Yaskawa INFORM job: R1_W27-A2(90,-90)POPR-KM-OK.JBI

/JOB
//NAME R1_W27-A2(90,-90)POPR-KM-OK
///FOLDERNAME KRIS-SCIANA
//POS
///NPOS 176,176,0,6,0,0
///TOOL 0
///POSTYPE PULSE
///PULSE
C00000=-47255,94033,21850,39667,98426,-85112
C00001=-10855,-90146,-90520,33531,76579,-85488
C00002=111602,-139984,-127808,5509,79015,30630
C00003=111602,-139984,-127808,5509,79015,30630
C00004=63451,-100439,-89596,34729,108559,18896
C00005=79235,-88636,-73634,36549,98880,22423
C00006=81155,-89027,-70716,36576,96440,22410
C00007=83679,-91038,-71523,36826,94925,22960
C00008=83320,-90762,-71414,36792,95139,22882
C00009=83320,-91266,-72707,36833,95574,23028
C00010=84421,-92107,-73039,36936,94918,23269
C00011=84421,-91766,-72172,36910,94628,23171
C00012=81728,-90820,-74480,36776,97327,22951
C00013=111602,-139984,-127808,5509,79015,30630
C00014=111602,-139984,-127808,5509,79015,30630
C00015=131748,-141997,-126846,-10495,77447,36936
C00016=120565,-130076,-92733,-8792,61450,34172
C00017=114295,-129242,-91918,-7183,60764,31836
C00018=112834,-127676,-89826,-6827,60159,31317
C00019=109595,-127191,-89697,-5944,60074,30085
C00020=111525,-128681,-91514,-6443,60572,30793
C00021=111525,-130307,-93896,-6407,61199,30757
C00022=120936,-129452,-91830,-16171,61520,34917
C00023=118478,-129412,-91819,-15577,61061,34026
C00024=114109,-131661,-95461,-7074,61680,31708
C00025=125724,-139860,-107023,-9755,65762,35760
C00026=168598,-161440,-97829,-65849,65951,-5239
C00027=139953,-89870,-86584,-36793,78283,-52428
C00028=129963,-49074,-62936,-33723,79499,-56916
C00029=128367,-48213,-57426,-33587,76404,-56612
C00030=128171,-46376,-53454,-33725,75068,-56281
C00031=127551,-46486,-53520,-33557,74812,-56456
C00032=127838,-49102,-55957,-33615,75055,-56414
C00033=127838,-49096,-59569,-33337,76927,-56985
C00034=130300,-24150,-34218,-41893,86298,-55823
C00035=130416,-25931,-34035,-41938,85581,-55484
C00036=130524,-27637,-35221,-41959,85519,-55412
C00037=130416,-25931,-34035,-41938,85581,-55484
C00038=129161,-28892,-39611,-41713,86429,-56383
C00039=125861,-39018,-45021,-41293,83456,-56659
C00040=125861,-38957,-44315,-41317,83150,-56538
C00041=125861,-39018,-45021,-41293,83456,-56659
C00042=132006,-10593,-25804,-42105,88453,-55942
C00043=125383,-9861,-27484,-30967,87136,-57090
C00044=124817,-9932,-27539,-30868,86930,-57252
C00045=125341,-12485,-30902,-30958,87772,-57281
C00046=124961,-12409,-32279,-30889,88403,-57596
C00047=121984,-15512,-34257,-30384,87021,-58359
C00048=122055,-13679,-30637,-30418,85927,-58040
C00049=122041,-11816,-29206,-30415,85989,-58061
C00050=122055,-13679,-30637,-30418,85927,-58040
C00051=122071,-15599,-34612,-30398,87201,-58373
C00052=118054,-13550,-32366,-29609,85516,-59451
C00053=118054,-13583,-31956,-29617,85281,-59389
C00054=118054,-13550,-32366,-29609,85516,-59451
C00055=125534,-18569,-39431,-41052,88700,-58862
C00056=123834,-57988,-65399,-23223,94284,39293
C00057=119710,-36131,-50756,-23492,104469,35737
C00058=119541,-35148,-48081,-23365,103369,35899
C00059=120820,-55138,-59718,-22945,91575,38721
C00060=119503,-55193,-60983,-22866,91905,38180
C00061=118759,-58952,-61759,-21710,87152,34499
C00062=120697,-55018,-60828,-22957,92227,38551
C00063=123778,-56814,-67966,-23331,96280,38880
C00064=80812,-71471,-83715,15937,85664,-13866
C00065=80812,-71834,-71790,16172,78419,-14815
C00066=107747,-97676,-64864,-15422,34839,20449
C00067=107974,-98087,-64546,-15779,34491,20660
C00068=108174,-97847,-63422,-16183,33983,20896
C00069=108174,-97847,-63422,-16183,33983,20896
C00070=109575,-108888,-72439,-17471,34149,21710
C00071=102046,-72347,-67920,-1263,67597,24279
C00072=76953,-69983,-67153,17125,77381,-16337
C00073=77709,-68021,-67434,16896,78355,-15929
C00074=96304,-74836,-69045,2706,67540,13944
C00075=85382,-70192,-66839,14096,72335,1446
C00076=83671,-68641,-66151,14549,72999,911
C00077=82927,-72320,-69596,14740,73354,686
C00078=82383,-44408,-60013,10514,90636,-51553
C00079=83267,-39109,-54206,10352,89686,-51335
C00080=93739,1438,-24878,6422,91479,-57500
C00081=93739,1438,-24878,6422,91479,-57500
C00082=93483,1925,-29171,6495,94374,-57435
C00083=103631,8716,-24589,-7355,104161,-72543
C00084=103148,15486,-14064,-7496,103326,-72736
C00085=105595,14163,-15273,-7551,103608,-71922
C00086=104864,13485,-18488,-6736,105180,-72257
C00087=101225,7871,-25887,-447,100429,-73560
C00088=94829,-40669,-100015,6490,88409,-74102
C00089=128133,-139556,-106944,-10306,66166,36618
C00090=113623,-140124,-95696,-7245,57468,31798
C00091=111191,-133211,-91671,-6501,58335,30798
C00092=112396,-117188,-87436,-6483,64023,30924
C00093=117788,-123916,-92276,-7889,64025,32937
C00094=117788,-143811,-128922,-7332,76251,32157
C00095=117788,-143811,-128922,-7332,76251,32157
C00096=-27890,68892,-2811,-32304,95656,-64919
C00097=-1389,132560,29341,8972,98096,-84314
C00098=-17183,121165,41486,39124,87360,-83411
C00099=45609,12223,-14680,25874,102540,-44378
C00100=55301,17182,-10314,25374,99523,-41463
C00101=55301,16672,-6013,25146,96878,-42036
C00102=55301,16639,-5464,25122,96557,-42106
C00103=55301,16672,-6013,25146,96878,-42036
C00104=52027,31709,8447,25239,96790,-43264
C00105=65662,27936,-1686,1783,97311,-42028
C00106=65925,27175,-1528,1759,96817,-41946
C00107=66144,26660,-2030,1742,96856,-41873
C00108=65925,27175,-1528,1759,96817,-41946
C00109=65925,27520,-3302,1766,98087,-41928
C00110=67752,27932,-3186,1610,98190,-41320
C00111=69686,29368,267,1433,96766,-40698
C00112=69239,27811,-1265,1472,96915,-40843
C00113=69714,29591,-377,1432,97275,-40681
C00114=70571,32771,2169,1358,97331,-40400
C00115=72811,38961,10399,1155,95415,-39677
C00116=73243,40763,12275,1116,95181,-39535
C00117=72717,38685,9237,1163,95989,-39704
C00118=70300,45171,15024,1377,95797,-40506
C00119=71840,46165,18079,1239,94403,-40008
C00120=72279,45156,17000,1201,94542,-39861
C00121=71840,46165,18079,1239,94403,-40008
C00122=71100,43306,13055,1308,96038,-40237
C00123=74981,35157,4595,968,97003,-38944
C00124=68153,50345,23565,13015,101581,-39746
C00125=68153,50336,23863,13003,101398,-39766
C00126=68153,50345,23565,13015,101581,-39746
C00127=74981,36365,46,979,100422,-38916
C00128=68608,6976,-17792,23795,112053,-53591
C00129=69057,8041,-13956,23524,110262,-53802
C00130=77166,501,-24156,13228,105180,-53608
C00131=69228,8608,-13543,23550,110248,-53738
C00132=68547,9857,-11185,23337,109691,-54121
C00133=80532,13332,-12849,13354,104269,-52437
C00134=69002,6644,-20376,25626,106012,-45957
C00135=36743,66838,47163,37250,103366,-40352
C00136=37959,59579,46469,37755,95211,-37788
C00137=37837,59881,47347,37721,94956,-37928
C00138=37624,60339,48596,37673,94623,-38135
C00139=36831,72187,58039,36474,100818,-41891
C00140=49145,73657,39688,12770,111067,-36167
C00141=47533,6238,-21702,16193,87850,-22319
C00142=48706,7477,-14718,15969,84101,-22409
C00143=50440,12407,-9463,15589,83099,-21944
C00144=49368,8705,-13714,15818,83988,-22197
C00145=48664,7312,-13691,15994,83418,-22513
C00146=49682,14586,-7490,15763,83149,-22198
C00147=45719,31490,8640,21979,89950,-33295
C00148=45824,34631,11803,21965,89613,-33319
C00149=48704,7662,-16449,15949,85218,-22264
C00150=47002,4841,-19925,16324,86209,-22716
C00151=51620,13344,-12650,-10356,82695,15963
C00152=52172,14147,-8973,-10543,80943,16297
C00153=53042,17284,-5127,-10797,80314,16646
C00154=52937,12849,-8980,-10764,80389,16602
C00155=52386,14618,-8611,-10600,80988,16365
C00156=54599,19555,-5413,-11177,81839,17037
C00157=52866,15720,-8829,-10712,81740,16462
C00158=52320,14787,-11359,-10544,82730,16194
C00159=103684,1413,-30862,2741,121345,77818
C00160=103850,2833,-28631,2757,120697,77864
C00161=102574,7420,-23963,2468,120223,77363
C00162=103907,3755,-28694,2786,121208,77898
C00163=104106,5504,-25931,2802,120401,77953
C00164=105308,5972,-25223,3052,120166,78404
C00165=104815,6248,-27488,2999,121717,78261
C00166=103683,1405,-30869,2741,121346,77818
C00167=103614,2055,-30742,3606,100061,77951
C00168=110138,-139455,-127658,5821,79297,30141
C00169=62576,-99046,-89073,34649,109242,18742
C00170=76661,-93546,-74524,35984,98364,21158
C00171=71402,-81532,-60843,44640,104085,20726
C00172=76616,-70399,-55778,46201,103281,22914
C00173=72927,-70202,-57613,45814,106055,22410
C00174=72965,-71329,-91142,53207,119453,30086
C00175=-4535,-93265,-111062,3717,101159,77715
BC00000=172948,1022366,1065683
BC00001=284631,1066333,1053590
BC00002=197512,1190309,1009585
BC00003=397680,1190309,1009585
BC00004=397680,1190309,1009585
BC00005=397680,1190309,1009585
BC00006=397680,1190309,1009585
BC00007=397680,1190309,1009585
BC00008=397680,1190309,1009585
BC00009=397680,1190309,1009585
BC00010=397680,1190309,1009585
BC00011=397680,1190309,1009585
BC00012=397680,1190309,1009585
BC00013=397680,1190309,1009585
BC00014=197512,1190309,1009585
BC00015=15680,1190309,1003705
BC00016=15680,1190309,1003705
BC00017=15680,1190309,1003705
BC00018=15680,1190309,1003705
BC00019=15680,1190309,1003705
BC00020=15680,1190309,1003705
BC00021=15680,1190309,1003705
BC00022=15680,1190309,1003705
BC00023=15680,1190309,1003705
BC00024=15680,1190309,1003705
BC00025=15680,1190309,1003705
BC00026=2250,1188982,1018188
BC00027=2245,1185181,1042831
BC00028=2245,1185181,1042831
BC00029=2245,1185181,1042831
BC00030=2245,1185181,1042831
BC00031=2245,1185181,1042831
BC00032=2245,1185181,1042831
BC00033=2245,1185181,1042831
BC00034=1991,1180873,1070755
BC00035=1991,1180873,1070755
BC00036=1991,1180873,1070755
BC00037=1991,1180873,1070755
BC00038=1991,1180873,1070755
BC00039=1991,1180873,1070755
BC00040=1991,1180873,1070755
BC00041=1991,1180873,1070755
BC00042=1991,1180873,1070755
BC00043=1991,1180873,1070755
BC00044=1991,1180873,1070755
BC00045=1991,1180873,1070755
BC00046=1991,1180873,1070755
BC00047=1991,1180873,1070755
BC00048=1991,1180873,1070755
BC00049=1991,1180873,1070755
BC00050=1991,1180873,1070755
BC00051=1991,1180873,1070755
BC00052=1991,1180873,1070755
BC00053=1991,1180873,1070755
BC00054=1991,1180873,1070755
BC00055=1991,1180873,1070755
BC00056=1991,1143594,1070910
BC00057=1991,1145344,1070910
BC00058=1991,1145344,1070910
BC00059=1991,1145344,1070910
BC00060=1991,1145344,1070910
BC00061=1991,1130616,1070910
BC00062=1991,1130116,1070910
BC00063=1991,1128866,1070910
BC00064=1991,1180480,1070910
BC00065=1991,1180480,1070910
BC00066=1992,1180480,1070906
BC00067=1992,1180480,1070906
BC00068=1992,1180480,1070906
BC00069=1992,1180480,1070906
BC00070=1992,1180480,1070906
BC00071=1992,1180480,1070906
BC00072=1991,1175938,1070910
BC00073=1991,1175938,1070910
BC00074=1992,1180480,1070906
BC00075=1992,1180480,1070906
BC00076=1992,1180480,1070906
BC00077=1992,1180480,1070906
BC00078=1992,1180480,1070906
BC00079=1993,1180480,1070905
BC00080=1992,1180480,1070906
BC00081=1992,1180480,1070906
BC00082=1992,1180480,1070906
BC00083=1993,1170260,1070904
BC00084=1993,1170260,1070902
BC00085=1993,1170260,1070902
BC00086=1993,1170260,1070904
BC00087=1992,1180480,1070906
BC00088=1992,1180480,1070906
BC00089=18069,1190309,1003705
BC00090=18069,1190309,1003705
BC00091=18069,1190309,1003705
BC00092=18069,1190309,1003705
BC00093=18069,1190309,1003705
BC00094=18069,1190309,1003705
BC00095=94851,1192591,1003705
BC00096=27006,1176774,1055878
BC00097=57075,1322294,1070892
BC00098=45628,1277740,1070896
BC00099=248889,1187650,1070910
BC00100=248889,1187650,1070910
BC00101=248889,1187650,1070910
BC00102=248889,1187650,1070910
BC00103=248889,1187650,1070910
BC00104=248889,1187650,1070910
BC00105=248889,1187650,1070910
BC00106=248889,1187650,1070910
BC00107=248889,1187650,1070910
BC00108=248889,1187650,1070910
BC00109=248889,1187650,1070910
BC00110=248889,1187650,1070910
BC00111=248889,1187650,1070910
BC00112=248889,1187650,1070910
BC00113=248889,1187650,1070910
BC00114=248889,1187650,1070910
BC00115=248889,1187650,1070910
BC00116=248889,1187650,1070910
BC00117=248889,1187650,1070910
BC00118=248889,1187650,1070910
BC00119=248889,1187650,1070910
BC00120=248889,1187650,1070910
BC00121=248889,1187650,1070910
BC00122=248889,1187650,1070910
BC00123=248889,1187650,1070910
BC00124=248889,1187650,1070910
BC00125=248889,1187650,1070910
BC00126=248889,1187650,1070910
BC00127=248889,1187650,1070910
BC00128=312191,1167362,1070910
BC00129=306535,1168545,1070910
BC00130=306538,1168544,1070910
BC00131=304272,1169019,1070910
BC00132=304272,1169019,1070910
BC00133=306538,1168544,1070910
BC00134=306535,1168545,1070910
BC00135=199299,1192678,1070910
BC00136=199299,1192678,1070910
BC00137=199299,1192678,1070910
BC00138=199299,1192678,1070910
BC00139=199299,1192678,1070910
BC00140=199299,1192678,1070910
BC00141=199962,1192678,1070910
BC00142=199962,1192678,1070910
BC00143=199962,1192678,1070910
BC00144=200228,1192678,1070910
BC00145=200228,1192678,1070910
BC00146=199962,1192678,1070910
BC00147=199962,1192678,1070910
BC00148=199962,1192678,1070910
BC00149=202074,1192678,1070910
BC00150=201410,1192678,1070910
BC00151=150763,1159292,1070910
BC00152=156327,1160542,1070910
BC00153=158126,1160946,1070907
BC00154=158552,1161042,1070910
BC00155=158552,1161042,1070910
BC00156=158692,1122943,1055155
BC00157=156466,1122443,1062648
BC00158=150903,1121193,1070910
BC00159=346682,1128113,1048282
BC00160=345916,1134373,1032919
BC00161=345708,1136079,1028733
BC00162=345610,1136877,1026774
BC00163=345610,1136877,1026774
BC00164=345708,1136079,1028733
BC00165=345610,1136877,1026774
BC00166=343614,1128095,1048354
BC00167=343613,1128096,1048352
BC00168=396087,1032525,1009585
BC00169=396087,1190309,1009585
BC00170=396087,1190309,1009585
BC00171=396087,1190309,1009585
BC00172=396087,1190309,1009585
BC00173=396087,1190309,1009585
BC00174=396087,1190309,1009585
BC00175=174979,687379,1048352
///POSTYPE BASE
///RECTAN
///RCONF 0,0,0,0,0,0,0,0,0,0,0,0,0,0,0,0,0,0,0,0,0,0,0,0
P00006=0.222,-3.123,-1.508,0.0000,0.0000,0.0000
P00023=0.143,-0.036,0.682,0.0000,0.0000,0.0000
P00024=0.145,-0.552,1.326,0.0000,0.0000,0.0000
P00025=-2.003,0.006,0.728,0.0000,0.0000,0.0000
P00040=-0.030,9.648,2.467,0.0000,0.0000,0.0000
P00041=0.192,3.924,0.305,0.0000,0.0000,0.0000
//INST
///DATE 2024/07/23 11:10
///ATTR SC,RW
///GROUP1 RB1,BS1
NOP
SFTOF
MOVJ C00000 BC00000 VJ=100.00
MOVJ C00001 BC00001 VJ=100.00
MOVJ C00002 BC00002 VJ=100.00
'DODANO BP 060624
MOVJ C00003 BC00003 VJ=100.00
MOVJ C00004 BC00004 VJ=100.00
MOVL C00005 BC00005 V=233.3
MOVL C00006 BC00006 V=60.0
REFP 3 C00007 BC00007
CALL JOB:SEARCH-R1
SET P040 P006
SFTON P040
MOVL C00008 BC00008 V=100.0
MOVL C00009 BC00009 V=100.0
MOVL C00010 BC00010 V=60.0
REFP 3 C00011 BC00011
CALL JOB:SEARCH-R1
SET P040 P006
SFTON P040
MOVL C00012 BC00012 V=100.0
SFTOF
MOVJ C00013 BC00013 VJ=100.00
MOVJ C00014 BC00014 VJ=100.00
MOVL C00015 BC00015 V=666.7
MOVL C00016 BC00016 V=666.7
MOVL C00017 BC00017 V=233.3
MOVL C00018 BC00018 V=60.0
REFP 3 C00019 BC00019
CALL JOB:SEARCH-R1
SET P041 P006
SFTON P041
MOVL C00020 BC00020 V=100.0
MOVL C00021 BC00021 V=100.0
MOVL C00022 BC00022 V=60.0
REFP 3 C00023 BC00023
CALL JOB:SEARCH-R1
SET P041 P006
SFTON P041
MOVL C00024 BC00024 V=100.0
MOVL C00025 BC00025 V=666.7
'KONIEC BP 060624
MOVJ C00026 BC00026 VJ=100.00
MOVJ C00027 BC00027 VJ=100.00
MOVJ C00028 BC00028 VJ=100.00
MOVJ C00029 BC00029 VJ=100.00
MOVL C00030 BC00030 V=60.0
REFP 3 C00031 BC00031
CALL JOB:SEARCH-R1
SET P023 P006
SFTON P023
MOVL C00032 BC00032 V=60.0
MOVL C00033 BC00033 V=100.0
MOVL C00034 BC00034 V=100.0
MOVL C00035 BC00035 V=100.0
REFP 3 C00036 BC00036
CALL JOB:SEARCH-R1
SET P023 P006
SFTON P023
MOVL C00037 BC00037 V=60.0
MOVL C00038 BC00038 V=100.0
MOVL C00039 BC00039 V=100.0
REFP 3 C00040 BC00040
CALL JOB:SEARCH-R1
SET P023 P006
SFTON P023
MOVL C00041 BC00041 V=60.0
'DRUGI NOWY POMIAR
SFTOF
MOVL C00042 BC00042 V=100.0
MOVL C00043 BC00043 V=100.0
REFP 3 C00044 BC00044
CALL JOB:SEARCH-R1
SET P024 P006
SFTON P024
MOVL C00045 BC00045 V=60.0
MOVL C00046 BC00046 V=100.0
MOVL C00047 BC00047 V=100.0
MOVL C00048 BC00048 V=60.0
REFP 3 C00049 BC00049
CALL JOB:SEARCH-R1
SET P024 P006
SFTON P024
MOVL C00050 BC00050 V=60.0
MOVL C00051 BC00051 V=100.0
MOVL C00052 BC00052 V=60.0
REFP 3 C00053 BC00053
CALL JOB:SEARCH-R1
SET P024 P006
SFTON P024
MOVL C00054 BC00054 V=60.0
MOVJ C00055 BC00055 VJ=30.00
SFTOF
'Path W988
SFTOF
SFTON P023
MOVJ C00056 BC00056 VJ=50.00
MOVJ C00057 BC00057 VJ=100.00
MOVL C00058 BC00058 V=100.0 PL=0
REFP 1 C00059 BC00059
REFP 2 C00060 BC00060
MACRO1 MJ#(0) ARGF7
ARCON
SFTON P024
MOVL C00061 BC00061 V=10.8
ARCOF
MOVL C00062 BC00062 V=100.0
MOVJ C00063 BC00063 VJ=50.00
SFTOF
'Path W989
SFTOF
SFTON P023
MOVJ C00064 BC00064 VJ=100.00
MOVJ C00065 BC00065 VJ=50.00
MOVL C00066 BC00066 V=100.0
ARCON
MOVL C00067 BC00067 V=8.3
MOVL C00068 BC00068 V=8.3
MOVL C00069 BC00069 V=8.3
ARCOF
SFTOF
MOVL C00070 BC00070 V=83.3
SFTON P023
MOVL C00071 BC00071 V=100.0 PL=0
REFP 1 C00072 BC00072
REFP 2 C00073 BC00073
MACRO1 MJ#(0) ARGF7
ARCON
TIMER T=0.50
MOVL C00074 BC00074 V=10.0
MOVL C00075 BC00075 V=10.0
MOVL C00076 BC00076 V=10.0
ARCOF
MOVJ C00077 BC00077 VJ=15.00
MOVJ C00078 BC00078 VJ=100.00
SFTON P023
MOVJ C00079 BC00079 VJ=100.00
ARCON
SFTON P024
MOVL C00080 BC00080 V=10.0
MOVL C00081 BC00081 V=10.0
ARCOF
MOVJ C00082 BC00082 VJ=15.00
MOVJ C00083 BC00083 VJ=100.00
MOVJ C00084 BC00084 VJ=20.00
ARCON
MOVL C00085 BC00085 V=10.0
ARCOF
MOVL C00086 BC00086 V=100.0
MOVL C00087 BC00087 V=166.7
MOVJ C00088 BC00088 VJ=100.00
SFTOF
'BP 060624
MOVJ C00089 BC00089 VJ=100.00
MOVJ C00090 BC00090 VJ=100.00
SFTON P041
MOVL C00091 BC00091 V=100.0 PL=0
MACRO1 MJ#(0) ARGF6
ARCON
MOVL C00092 BC00092 V=12.5
ARCOF
MOVL C00093 BC00093 V=11.7
SFTOF
MOVL C00094 BC00094 V=666.7
MOVL C00095 BC00095 V=666.7
'KONIEC BP 060624
'2 STRONA
MOVJ C00096 BC00096 VJ=100.00
'Path VIA1124
SFTOF
MOVJ C00097 BC00097 VJ=100.00
CALL JOB:ONLY_CUT_KM_NEW_SCIANA
'Path S992
SFTOF
MOVJ C00098 BC00098 VJ=100.00
SFTOF
MOVJ C00099 BC00099 VJ=100.00
MOVJ C00100 BC00100 VJ=100.00
MOVL C00101 BC00101 V=133.3
REFP 3 C00102 BC00102
CALL JOB:SEARCH-R1
SET P024 P006
SFTON P024
MOVL C00103 BC00103 V=60.0
MOVL C00104 BC00104 V=100.0
MOVL C00105 BC00105 V=100.0
MOVL C00106 BC00106 V=100.0
REFP 3 C00107 BC00107
CALL JOB:SEARCH-R1
SET P024 P006
SFTON P024
MOVL C00108 BC00108 V=60.0
MOVL C00109 BC00109 V=250.0
MOVL C00110 BC00110 V=250.0
MOVL C00111 BC00111 V=166.7
REFP 3 C00112 BC00112
CALL JOB:SEARCH-R1
SET P024 P006
SFTON P024
MOVL C00113 BC00113 V=333.3
SFTOF
MOVL C00114 BC00114 V=250.0
MOVL C00115 BC00115 V=166.7
REFP 3 C00116 BC00116
CALL JOB:SEARCH-R1
SET P025 P006
SFTON P025
MOVL C00117 BC00117 V=250.0
MOVL C00118 BC00118 V=333.3
MOVL C00119 BC00119 V=250.0
REFP 3 C00120 BC00120
CALL JOB:SEARCH-R1
SET P025 P006
SFTON P025
MOVL C00121 BC00121 V=250.0
MOVL C00122 BC00122 V=250.0
MOVL C00123 BC00123 V=333.3
MOVL C00124 BC00124 V=166.7
REFP 3 C00125 BC00125
CALL JOB:SEARCH-R1
SET P025 P006
SFTON P025
MOVL C00126 BC00126 V=166.7
MOVL C00127 BC00127 V=333.3
'Path W993
SFTOF
SFTON P024
MOVJ C00128 BC00128 VJ=100.00
MOVJ C00129 BC00129 VJ=100.00
SFTON P024
MOVL C00130 BC00130 V=100.0 PL=0
REFP 1 C00131 BC00131
REFP 2 C00132 BC00132
MACRO1 MJ#(0) ARGF7
ARCON
SFTON P025
MOVL C00133 BC00133 V=10.0
ARCOF
MOVL C00134 BC00134 V=166.7
SFTOF
SFTON P024
MOVJ C00135 BC00135 VJ=20.00
MOVJ C00136 BC00136 VJ=20.00
ARCON
MOVL C00137 BC00137 V=8.3
MOVL C00138 BC00138 V=8.3
ARCOF
MOVL C00139 BC00139 V=416.7
MOVJ C00140 BC00140 VJ=20.00
MOVJ C00141 BC00141 VJ=20.00
MOVJ C00142 BC00142 VJ=100.00
SFTON P024
MOVL C00143 BC00143 V=100.0 PL=0
REFP 1 C00144 BC00144
REFP 2 C00145 BC00145
MACRO1 MJ#(0) ARGF7
ARCON
MOVL C00146 BC00146 V=10.0
MOVL C00147 BC00147 V=10.0
MOVL C00148 BC00148 V=10.0
ARCOF
MOVL C00149 BC00149 V=100.0
MOVL C00150 BC00150 V=166.7
SFTOF
'Path W995
SFTOF
SFTON P024
MOVJ C00151 BC00151 VJ=100.00
MOVJ C00152 BC00152 VJ=100.00
SFTON P024
MOVL C00153 BC00153 V=100.0 PL=0
REFP 1 C00154 BC00154
REFP 2 C00155 BC00155
MACRO1 MJ#(0) ARGF7
ARCON
SFTON P025
MOVL C00156 BC00156 V=10.0
ARCOF
MOVL C00157 BC00157 V=400.0
MOVL C00158 BC00158 V=1000.0
SFTOF
MOVJ C00159 BC00159 VJ=100.00
MOVJ C00160 BC00160 VJ=100.00
SFTON P025
MOVL C00161 BC00161 V=166.7 PL=0
REFP 1 C00162 BC00162
REFP 2 C00163 BC00163
MACRO1 MJ#(0) ARGF7
ARCON
MOVL C00164 BC00164 V=10.0
ARCOF
MOVL C00165 BC00165 V=166.7
MOVL C00166 BC00166 V=166.7
SFTOF
MOVJ C00167 BC00167 VJ=100.00
'BP 060624
SFTOF
MOVL C00168 BC00168 V=666.7
MOVL C00169 BC00169 V=666.7
MOVL C00170 BC00170 V=666.7
SFTON P040
MOVL C00171 BC00171 V=100.0 PL=0
MACRO1 MJ#(0) ARGF6
ARCON
MOVL C00172 BC00172 V=12.5
ARCOF
MOVL C00173 BC00173 V=266.7
SFTOF
MOVJ C00174 BC00174 VJ=100.00
'KONIEC BP 060624
MOVJ C00175 BC00175 VJ=100.00
END
